# EPICS alarm handler configuration: alh_files/mgnt_li22_lgps.alhConfig
GROUP NULL LGPS:LI22:MG01
$ALIAS LGPS
$GUIDANCE
LI22 LGPS magnets
   Group Name: LGPS:LI22:MG01
   Summary PV:  LGPS:LI22:MG01:STATSUMY
$END

GROUP LGPS:LI22:MG01  LGPS:LI22:2
CHANNEL     LGPS:LI22:2           LGPS:LI22:2:STATMSG   -----
   $FORCEPV LGPS:LI22:2:STATMSGSV -DATL 1 0
